Staubli VAL3: getPoint.pgx

public program getPoint(trsf& x_trPoint, string x_sPallet)
begin
end
